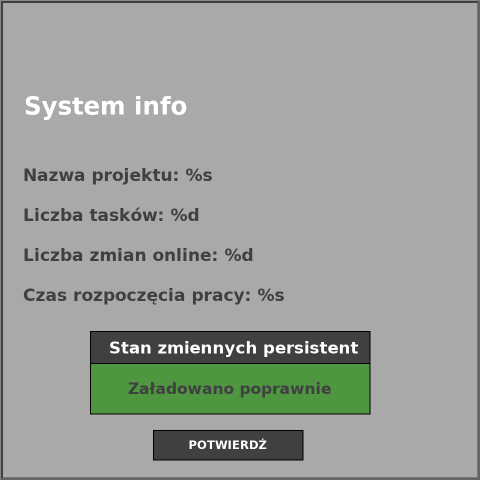
VISUALIZATION PH_SystemInfo  // 480x480
VAR
	bConfirmButtonState						: BOOL:=FALSE;
END_VAR
    Rectangle (0,0 480x480)
    Rectangle (90,331 280x83)
    Label (21,91 175x30), "System info"
    Rectangle (20,160 339x30), "Nazwa projektu: %s", text variable: _AppInfo.ProjectName
    Rectangle (20,200 339x30), "Liczba tasków: %d", text variable: _AppInfo.TaskCnt
    Rectangle (20,240 339x30), "Liczba zmian online: %d", text variable: _AppInfo.OnlineChangeCnt
    Rectangle (20,280 437x30), "Czas rozpoczęcia pracy: %s", text variable: P_SystemInfo.sStartTime
    RoundedRectangle (153,430 150x30), "POTWIERDŹ", colour toggle: bConfirmButtonState
        OnMouseUp: execute { bConfirmButtonState:=FALSE; }
        OnMouseUp: execute { P_SystemInfo.bConfirm:=FALSE; }
        OnMouseLeave: execute { bConfirmButtonState:=FALSE; }
        OnMouseLeave: execute { P_SystemInfo.bConfirm:=FALSE; }
        OnMouseDown: execute { bConfirmButtonState:=TRUE; }
        OnMouseDown: execute { P_SystemInfo.bConfirm:=TRUE; }
    Rectangle (95,333 258x30), "Stan zmiennych persistent"
    Rectangle (90,363 280x51), "Błąd", invisible if: NOT P_SystemInfo.bError
    Rectangle (90,363 280x51), "Załadowano plik zapasowy", invisible if: NOT P_SystemInfo.bWarning
    Rectangle (90,363 280x51), "Załadowano poprawnie", invisible if: NOT P_SystemInfo.bOK
END_VISUALIZATION

(* stored: Version 1.1.0.1, ProductVersion 3.1.4024.3
   Visu PH_SystemInfo: Id {7741d480-7938-44cd-9497-98a724698d6e} *)
